// TIA Portal V19 export
TYPE "CTrk_Item"
// stored: Access Published
   STRUCT
      C_ID : DInt;   // ID coil
      DecoilerX : SInt;
      MES_CN : DInt;   // MES : Numeo identificatico bobina
      MES_HN : DInt;   // MES: Numero di colata
      Provino_Req : SInt;
      Provino_Done : SInt;
      Loaded : "CTrk_Log";   // Materiale è stato caricato (nel mandrino dell'aspo)
      Processing : Array[1..20] of "CTrk_Log";   // Materiale è in lavorazione
      Consumed : "CTrk_Log";   // Materiale concluso (fine coil)
      Interrupted : "CTrk_Log";   // Interruzione uso del materiale in lavoro (taglio per rimuoverlo / per fare provino)
   END_STRUCT;
END_TYPE
